TYPE
	MF_INDEX : INT;
END_TYPE

(* stored: Version 1.1.0.1, ProductVersion 3.1.4024.6
   DUT MF_INDEX: Id {5ff9f34b-b6d4-4e3b-9be8-3f33c2e220f7} *)
